Staubli VAL3: IoWriteRequest.dtx

public num nCount
public num nType
public num nIndex
public num nValue
